Universal Robots PolyScope program: tele1.urp

Program tele1 (installation=default directory=/programs createdIn=5.9.1.1031110 lastSavedIn=5.9.1.1031110 robotSerialNumber=20195501059)
Calibrated DH parameters: a=[0.000146, -0.418764, -0.053981, 0.000058, -0.000023, 0]; d=[0.162545, 37.319448, -206.067439, 168.881546, 0.09955, 0.099464]; alpha=[1.57004, -0.001979, 0.002304, 1.570607, -1.57066, 0]; deltaTheta=[0, -0.174616, -1.258233, 1.432844, -0.000001, 0]
Robot Program (runOnlyOnce=false)
  MoveJ speed 60 deg/s, acceleration 80 deg/s^2 (useActiveTCP=true) feature=Base
    Waypoint Waypoint_1: TCP in base x=219.845 y=-479.76 z=63.752 mm, rx=-2.1225 ry=-2.2569 rz=0.2476 rad; joints [104.563, -76.335, 115.445, -132.359, 261.289, -259.164] deg; TCP offset x=0 y=0 z=174 mm, rx=0 ry=0 rz=0 rad
  MoveL speed 250 mm/s, acceleration 1200 mm/s^2 (useActiveTCP=true) feature=Base
    Waypoint Waypoint_2: TCP in base x=219.84 y=-357.579 z=63.753 mm, rx=-2.1225 ry=-2.2568 rz=0.2476 rad; joints [109.072, -89.605, 130.765, -133.705, 261.089, -254.601] deg
    URCap Olis Teleop (Olis Teleop, Olis Robotics) dataModel(OperatorMessage=Time for Teleop!)
    Waypoint Waypoint_1: TCP in base x=219.845 y=-479.76 z=63.752 mm, rx=-2.1225 ry=-2.2569 rz=0.2476 rad; joints [104.563, -76.335, 115.445, -132.359, 261.289, -259.164] deg
